FUNCTION_BLOCK FB112
TITLE = 'pilot'
AUTHOR : CB

VAR
	pilot_F1 : FB93;
	pilot_F2 : FB102;
	pilot_F3 : FB110;
END_VAR


BEGIN


NETWORK
TITLE =
//
//	pilot/pilot_F1
CALL #pilot_F1;



NETWORK
TITLE =
//
//	pilot/pilot_F2
CALL #pilot_F2;



NETWORK
TITLE =
//
//	pilot/pilot_F3
CALL #pilot_F3;




END_FUNCTION_BLOCK
